INTERFACE I_ComponentBase_SR

END_INTERFACE

(* stored: Version 1.1.0.1
   Itf I_ComponentBase_SR: Id {419a3803-847e-4542-9981-d24c68184140} *)
